PROGRAM Funcs
VAR
END_VAR

END_PROGRAM

(* stored: Version 1.1.0.1, ProductVersion 3.1.4024.12
   POU Funcs: Id {ee771c61-4cc8-49fe-a213-1138bcc939e9}, SpecialFunc None *)
